TYPE M2Statuses :
STRUCT
	initializationStatus: InitializationStatus;
	poweredStatus: PoweredStatus;
	healthStatus: HealthStatus;
	busyStatus: BusyStatus;
	operatingStatus: OperatingStatus;
END_STRUCT
END_TYPE

(* stored: Version 1.1.0.1, ProductVersion 3.1.4019.2
   DUT M2Statuses: Id {0ce72105-fcb9-41c5-9251-522d63440389} *)
